# EPICS substitutions: vme_iocs/iocbio4/iocBoot/UNUSED/fb_epid.substitutions
# $Id: fb_epid.substitutions 14505 2012-02-29 21:25:07Z jemian $

file "$(OPTICS)/opticsApp/Db/fb_epid.db"
  {
    {
        P=18IDd:epid1,
	IN=18IDd:epid1:sim.VAL,
	OUT=18IDd:epid1:sim.D,
	MODE=PID,
	CALC=A,
	PERMIT1="18IDd:epid1:on.VAL",
	PERMIT2="",
	PERMIT3="",
	PERMIT4=""
    }
  }
